TYPE E_RejectPanelState :
(
	INIT,
	EMPTY,
	OCCUPIED,
	ERROR
);
END_TYPE

(* stored: Version 1.1.0.1, ProductVersion 3.1.4022.12
   DUT E_RejectPanelState: Id {9fab34e2-905a-42bf-855c-69224b8301ab} *)
